    |   movel(pose_trans(ref_frame,p[0.023213, 0.134859, -0.000125, -0.013708, 3.141563, 0.000000]),accel_mss,speed_ms,0,0.001)
    |   movel(pose_trans(ref_frame,p[0.024024, 0.134865, -0.000125, -0.013708, 3.141563, -0.000000]),accel_mss,speed_ms,0,0.001)
    |   movel(pose_trans(ref_frame,p[0.024029, 0.135970, -0.000125, -0.013708, 3.141563, -0.000000]),accel_mss,speed_ms,0,0.001)
    |   movel(pose_trans(ref_frame,p[0.024034, 0.137075, -0.000125, -0.013708, 3.141563, 0.000000]),accel_mss,speed_ms,0,0.001)
    |   movel(pose_trans(ref_frame,p[0.022932, 0.137075, -0.000125, -0.013708, 3.141563, 0.000000]),accel_mss,speed_ms,0,0.001)
    |   movel(pose_trans(ref_frame,p[0.021829, 0.137075, -0.000125, -0.013708, 3.141563, 0.000000]),accel_mss,speed_ms,0,0.001)
    |   movel(pose_trans(ref_frame,p[0.021877, 0.136331, -0.000125, -0.013708, 3.141563, 0.000000]),accel_mss,speed_ms,0,0.001)
    |   movel(pose_trans(ref_frame,p[0.021890, 0.135997, -0.000125, -0.013708, 3.141563, -0.000000]),accel_mss,speed_ms,0,0.001)
    |   movel(pose_trans(ref_frame,p[0.021886, 0.135664, -0.000125, -0.013708, 3.141563, -0.000000]),accel_mss,speed_ms,0,0.001)
    |   movel(pose_trans(ref_frame,p[0.021855, 0.135492, -0.000125, -0.013708, 3.141563, 0.000000]),accel_mss,speed_ms,0,0.001)
    |   movel(pose_trans(ref_frame,p[0.021777, 0.135336, -0.000125, -0.013708, 3.141563, 0.000000]),accel_mss,speed_ms,0,0.001)
    |   movel(pose_trans(ref_frame,p[0.021666, 0.135228, -0.000125, -0.013708, 3.141563, 0.000000]),accel_mss,speed_ms,0,0.001)
    |   movel(pose_trans(ref_frame,p[0.021524, 0.135169, -0.000125, -0.013708, 3.141563, 0.000000]),accel_mss,speed_ms,0,0.001)
    |   movel(pose_trans(ref_frame,p[0.021277, 0.135130, -0.000125, -0.013708, 3.141563, -0.000000]),accel_mss,speed_ms,0,0.001)
    |   movel(pose_trans(ref_frame,p[0.021026, 0.135115, -0.000125, -0.013708, 3.141563, 0.000000]),accel_mss,speed_ms,0,0.001)
    |   movel(pose_trans(ref_frame,p[0.020896, 0.135115, -0.000125, -0.013708, 3.141563, 0.000000]),accel_mss,speed_ms,0,0.001)
    |   movel(pose_trans(ref_frame,p[0.020766, 0.135121, -0.000125, -0.013708, 3.141563, 0.000000]),accel_mss,speed_ms,0,0.001)
    |   movel(pose_trans(ref_frame,p[0.020646, 0.135130, -0.000125, -0.013708, 3.141563, 0.000000]),accel_mss,speed_ms,0,0.001)
    |   movel(pose_trans(ref_frame,p[0.020527, 0.135145, -0.000125, -0.013708, 3.141563, 0.000000]),accel_mss,speed_ms,0,0.001)
    |   movel(pose_trans(ref_frame,p[0.020430, 0.135161, -0.000125, -0.013708, 3.141563, -0.000000]),accel_mss,speed_ms,0,0.001)
    |   movel(pose_trans(ref_frame,p[0.020333, 0.135181, -0.000125, -0.013708, 3.141563, 0.000000]),accel_mss,speed_ms,0,0.001)
    |   movel(pose_trans(ref_frame,p[0.020288, 0.135199, -0.000125, -0.013708, 3.141563, 0.000000]),accel_mss,speed_ms,0,0.001)
    |   movel(pose_trans(ref_frame,p[0.020249, 0.135228, -0.000125, -0.013708, 3.141563, 0.000000]),accel_mss,speed_ms,0,0.001)
    |   movel(pose_trans(ref_frame,p[0.020218, 0.135270, -0.000125, -0.013708, 3.141563, -0.000000]),accel_mss,speed_ms,0,0.001)
    |   movel(pose_trans(ref_frame,p[0.020202, 0.135319, -0.000125, -0.013708, 3.141563, -0.000000]),accel_mss,speed_ms,0,0.001)
    |   movel(pose_trans(ref_frame,p[0.020183, 0.135442, -0.000125, -0.013708, 3.141563, -0.000000]),accel_mss,speed_ms,0,0.001)
    |   movel(pose_trans(ref_frame,p[0.020167, 0.135567, -0.000125, -0.013708, 3.141563, -0.000000]),accel_mss,speed_ms,0,0.001)
    |   movel(pose_trans(ref_frame,p[0.020153, 0.135719, -0.000125, -0.013708, 3.141563, -0.000000]),accel_mss,speed_ms,0,0.001)
    |   movel(pose_trans(ref_frame,p[0.020145, 0.135872, -0.000125, -0.013708, 3.141563, -0.000000]),accel_mss,speed_ms,0,0.001)
    |   movel(pose_trans(ref_frame,p[0.020141, 0.136041, -0.000125, -0.013708, 3.141563, -0.000000]),accel_mss,speed_ms,0,0.001)
    |   movel(pose_trans(ref_frame,p[0.020141, 0.136210, -0.000125, -0.013708, 3.141563, 0.000000]),accel_mss,speed_ms,0,0.001)
    |   movel(pose_trans(ref_frame,p[0.020155, 0.137072, -0.000125, -0.013708, 3.141563, -0.000000]),accel_mss,speed_ms,0,0.001)
    |   movel(pose_trans(ref_frame,p[0.019067, 0.137076, -0.000125, -0.013708, 3.141563, 0.000000]),accel_mss,speed_ms,0,0.001)
    |   movel(pose_trans(ref_frame,p[0.017979, 0.137081, -0.000125, -0.013708, 3.141563, -0.000000]),accel_mss,speed_ms,0,0.001)
    |   movel(pose_trans(ref_frame,p[0.017974, 0.136223, -0.000125, -0.013708, 3.141563, -0.000000]),accel_mss,speed_ms,0,0.001)
    |   movel(pose_trans(ref_frame,p[0.017971, 0.136054, -0.000125, -0.013708, 3.141563, -0.000000]),accel_mss,speed_ms,0,0.001)
    |   movel(pose_trans(ref_frame,p[0.017963, 0.135886, -0.000125, -0.013708, 3.141563, 0.000000]),accel_mss,speed_ms,0,0.001)
    |   movel(pose_trans(ref_frame,p[0.017951, 0.135733, -0.000125, -0.013708, 3.141563, -0.000000]),accel_mss,speed_ms,0,0.001)
    |   movel(pose_trans(ref_frame,p[0.017934, 0.135581, -0.000125, -0.013708, 3.141563, 0.000000]),accel_mss,speed_ms,0,0.001)
    |   movel(pose_trans(ref_frame,p[0.017916, 0.135457, -0.000125, -0.013708, 3.141563, -0.000000]),accel_mss,speed_ms,0,0.001)
    |   movel(pose_trans(ref_frame,p[0.017894, 0.135334, -0.000125, -0.013708, 3.141563, 0.000000]),accel_mss,speed_ms,0,0.001)
    |   movel(pose_trans(ref_frame,p[0.017877, 0.135285, -0.000125, -0.013708, 3.141563, 0.000000]),accel_mss,speed_ms,0,0.001)
    |   movel(pose_trans(ref_frame,p[0.017846, 0.135243, -0.000125, -0.013708, 3.141563, -0.000000]),accel_mss,speed_ms,0,0.001)
    |   movel(pose_trans(ref_frame,p[0.017804, 0.135212, -0.000125, -0.013708, 3.141563, 0.000000]),accel_mss,speed_ms,0,0.001)
    |   movel(pose_trans(ref_frame,p[0.017755, 0.135194, -0.000125, -0.013708, 3.141563, 0.000000]),accel_mss,speed_ms,0,0.001)
    |   movel(pose_trans(ref_frame,p[0.017631, 0.135173, -0.000125, -0.013708, 3.141563, -0.000000]),accel_mss,speed_ms,0,0.001)
    |   movel(pose_trans(ref_frame,p[0.017507, 0.135155, -0.000125, -0.013708, 3.141563, 0.000000]),accel_mss,speed_ms,0,0.001)
    |   movel(pose_trans(ref_frame,p[0.017355, 0.135138, -0.000125, -0.013708, 3.141563, 0.000000]),accel_mss,speed_ms,0,0.001)
    |   movel(pose_trans(ref_frame,p[0.017203, 0.135126, -0.000125, -0.013708, 3.141563, -0.000000]),accel_mss,speed_ms,0,0.001)
    |   movel(pose_trans(ref_frame,p[0.017034, 0.135118, -0.000125, -0.013708, 3.141563, 0.000000]),accel_mss,speed_ms,0,0.001)
    |   movel(pose_trans(ref_frame,p[0.016865, 0.135115, -0.000125, -0.013708, 3.141563, 0.000000]),accel_mss,speed_ms,0,0.001)
    |   movel(pose_trans(ref_frame,p[0.016008, 0.135109, -0.000125, -0.013708, 3.141563, -0.000000]),accel_mss,speed_ms,0,0.001)
    |   movel(pose_trans(ref_frame,p[0.016011, 0.134006, -0.000125, -0.013708, 3.141563, 0.000000]),accel_mss,speed_ms,0,0) # end trace
    |   speed_ms    = 1.000
    |   movel(pose_trans(ref_frame,p[0.016011, 0.134006, 0.005000, -0.013708, 3.141563, 0.000000]),accel_mss,speed_ms,0,0.001)
    |   movel(pose_trans(ref_frame,p[0.000000, 0.000000, 0.005000, -0.013708, 3.141563, -0.000000]),accel_mss,speed_ms,0,0.001)
    |   movel(pose_trans(ref_frame,p[0.000000, 0.000000, 0.055000, -0.013708, 3.141563, -0.000000]),accel_mss,speed_ms,0,0.001)
    |   # End of main program
    | end
    | 
    | output_RSettings()
  Halt
